FUNCTION_BLOCK FB_AnalogInput
VAR_INPUT
END_VAR
VAR_INPUT
	nValue				: INT; //input value
END_VAR
VAR_OUTPUT
	fValue 				: REAL; //converted value
END_VAR
VAR
	fUpperLimit : REAL; //upper limit of value range
	fLowerLimit : REAL; //lower limit of value range
END_VAR

// conversion from Bit value to actual value
fValue := ((INT_TO_REAL(nValue) / 32767 * (fUpperLimit - fLowerLimit)) + fLowerLimit);

METHOD FB_init : BOOL
VAR_INPUT
	bInitRetains : BOOL; // if TRUE, the retain variables are initialized (warm start / cold start)
	bInCopyCode : BOOL;  // if TRUE, the instance afterwards gets moved into the copy code (online change)
	fUpperLimit : REAL; //upper limit of value range
	fLowerLimit : REAL; //lower limit of value range
END_VAR
//copy input values to internal variables
THIS^.fUpperLimit := fUpperLimit;
THIS^.fLowerLimit := fLowerLimit;
END_METHOD

END_FUNCTION_BLOCK

(* stored: Version 1.1.0.1, ProductVersion 3.1.4024.9
   POU FB_AnalogInput: Id {974da21a-71f8-4eb5-a649-07e9e0dfb2bc}, SpecialFunc None
   Method FB_init: Id {de7075cb-1aef-489c-8a92-b92c57b0d4d5} *)
